{attribute 'OPC.UA.DA' := '1'}
{attribute 'OPC.UA.DA.StructuredType' := '1'}
{attribute 'pack_mode' := '1'}
TYPE ST_Complex_4 :
STRUCT
	ErrorID : E_Enum_1;
END_STRUCT
END_TYPE

(* stored: Version 1.1.0.1
   DUT ST_Complex_4: Id {da197fd3-f0c3-45f5-a0f1-8e7a177e04bf} *)
